Xinje XDPPro project, PLC1: XDH-60A32 (software 3.8.0a 2025-04-30)

PROGRAM 梯形图

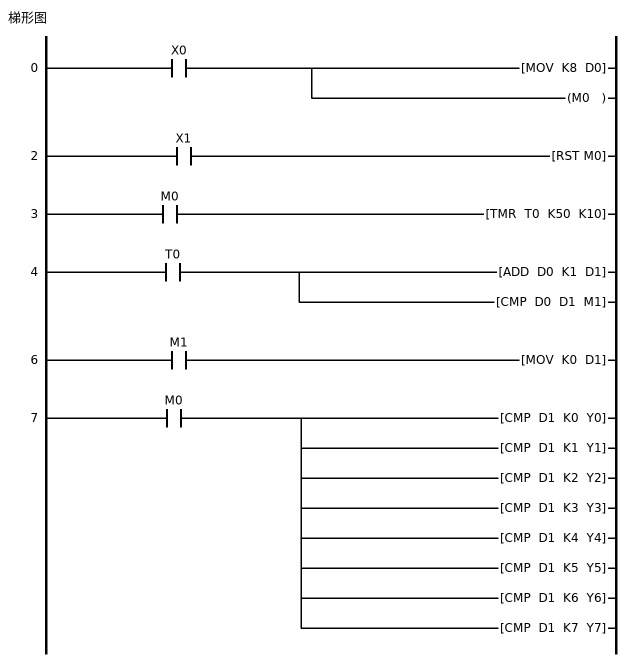
LD     X0
MOV    K8 D0
OUT    M0
LD     X1
RST    M0
LD     M0
TMR    T0 K50 K10
LD     T0
ADD    D0 K1 D1
CMP    D0 D1 M1
LD     M1
MOV    K0 D1
LD     M0
CMP    D1 K0 Y0
CMP    D1 K1 Y1
CMP    D1 K2 Y2
CMP    D1 K3 Y3
CMP    D1 K4 Y4
CMP    D1 K5 Y5
CMP    D1 K6 Y6
CMP    D1 K7 Y7